{attribute 'qualified_only'}
{attribute 'strict'}
{attribute 'to_string'}
TYPE E_RackFeederCmd :
(
	noCmd := 0,
	TeachTrolleyDock,
	TeachStorageDock
);
END_TYPE

(* stored: Version 1.1.0.1
   DUT E_RackFeederCmd: Id {88efeaf1-30e4-4786-bc9e-94a70d5b5bc7} *)
